(* CODESYS project PiecuchProjekt.export

Project tree, tasks and I/O mapping:
  Device : CODESYS Control Win V3, 3S - Smart Software Solutions GmbH, version 3.5.16.40
    application Application
      libraries: Standard, * (System)
      task MainTask (cyclic, interval t#20ms, priority 1) calls PLC_PRG
      global variables HMI
      global variables OPC
      program PLC_PRG [ST]
      function block TwoAxisLogic [ST]
*)

// Device/Application/HMI
{attribute 'qualified_only'}
VAR_GLOBAL
	GoingQA : BOOL;
	Emitter1Color : INT;
	Emitter2Color : INT;
END_VAR

// Device/Application/OPC
{attribute 'qualified_only'}
VAR_GLOBAL
	// This part includes 2 first machines center and surroundings machines
	iAtAssembledConvEntry : BOOL;
	iAtAssemledPosition : BOOL;
	iMachine1Exit : BOOL;
	iMachine2Exit : BOOL;
	iMachine1Entry : BOOL;
	iMachine2Entry : BOOL;
	iMachiningCenter1Error : BOOL;
	iMachiningCenter2Error : BOOL;
	iMachiningCenter1IsBusy : BOOL;
	iMachiningCenter1Opened : BOOL;
	iMachiningCenter2IsBusy : BOOL;
	iMachiningCenter2Opened : BOOL;
	iMachiningCenter1Progress : INT;
	iMachiningCenter2Progress : INT;
	iRightPositioner2Clamped : BOOL;
	iRightPositioner1Clamped : BOOL;
	iRightPositioner1OnPlace : BOOL;
	iRightPositioner2OnPlace : BOOL;
	iRightPositioner3Clamped : BOOL;
	iRightPositioner3OnPlace : BOOL;
	iTwoAxis1Grabbed : BOOL;
	iTwoAxis1MovingX : BOOL;
	iTwoAxis1MovingZ : BOOL;
	iVisionSenserPart1 : INT;
	iVisionSenserPart2 : INT;
	
	oAssembledMaterialConv : BOOL;
	oBaseMaterialConv1 : BOOL;
	oBaseMaterialConv2 : BOOL;
	oEmitter1Base : INT;
	oEmitter1Emit : BOOL;
	oEmitter1Part : INT;
	oEmitter2Base : INT;
	oEmitter2Emit : BOOL;
	oEmitter2Part : INT;
	oLiquidMaterialConv1 : BOOL;
	oLiquidMaterialConv2 : BOOL;
	oMachiningCenter1Product : BOOL;
	oMachiningCenter2Product : BOOL;
	oRawMaterialSupply1 : BOOL;
	oRawMaterialSupply2 : BOOL;
	oRightPositioner2Clamp : BOOL;
	oRightPositioner1Clamp : BOOL;
	oRightPositioner1Raise : BOOL;
	oRightPositioner2Raise : BOOL;
	oRightPositioner3Clamp : BOOL;
	oRightPositioner3Raise : BOOL;
	oTwoAxis1X : BOOL;
	oTwoAxis1Z : BOOL;
	oTwoAxis1Grab : BOOL;
	
	//This part include second and third twoAxis pick and place, QA and surroundings conveyors, and first warehouse conveyros
	iAtAssemblyLoadEntry : BOOL;
	iAtCrane1Entry : BOOL;
	iAtCurveConv1Exit : BOOL;
	iAtCurveConv1Entry : BOOL;
	iAtFirstwarehouseCurveConv2Exit : BOOL;
	iAtFirstwarehouseCurveConv2Entry : BOOL;
	iAtPusher : BOOL;
	iAtQACurveEntry : BOOL;
	iAtQAEntry : BOOL;
	iAtQAExit : BOOL;
	iAtWeightConvExit : BOOL;
	iAtWeightConvEntry : BOOL;
	iAtTurntable1Entry : BOOL;
	iAtTurntable1ExitQA : BOOL;
	iAtTurntable1ExitNormal : BOOL;
	iPusher1Back : BOOL;
	iPusher2Back : BOOL;
	iPusher3Back : BOOL;
	iPusher1Front : BOOL;
	iPusher2Front : BOOL;
	iPusher3Front : BOOL;
	iTurntable1Back : BOOL;
	iTurntable1Front : BOOL;
	iTurntable1AtZero : BOOL;
	iTurntable1AtNinety : BOOL;
	iTwoAxis2Grabbed : BOOL;
	iTwoAxis2MovingX : BOOL;
	iTwoAxis3Grabbed : BOOL;
	iTwoAxis3MovingX : BOOL;
	iTwoAxis3MovingZ : BOOL;
	iTwoAxis2MovingZ : BOOL;
	iVisionSensor1 : BOOL;
	iVisionSensor2 : BOOL;
	iWeightConv : REAL;
	iAtQALightConvExit : BOOL;
	
	oFirstWarehouseConv1 : BOOL;
	oFirstWarehouseConv3 : BOOL;
	oFirstWarehouseConvLoad : BOOL;
	oFirstWarehouseCurveConv2 : BOOL;
	oPalletAndBoxConv1 : BOOL;
	oPalletAndBoxConv3 : BOOL;
	oPalletAndBoxCurveConv2 : BOOL;
	oPusher1 : BOOL;
	oPusher2 : BOOL;
	oPusher3 : BOOL;
	oQAConv : BOOL;
	oQACurveConv : BOOL;
	oQALightConv1 : BOOL;
	oQALightConv2 : BOOL;
	oQALightConv3 : BOOL;
	oQALightConv4 : BOOL;
	oTurntable1Turn : BOOL;
	oTurntable1Forward : BOOL;
	oTurntable1Backward : BOOL;
	oTwoAxis2X : BOOL;
	oTwoAxis2Z : BOOL;
	oTwoAxis3X : BOOL;
	oTwoAxis3Z : BOOL;
	oTwoAxis2Grab : BOOL;
	oTwoAxis3Grab : BOOL;
	oWeightConvBackward : BOOL;
	oWeightConvToward : BOOL;
	
	//This part includes two cranes and conveyor betweeen them
	iAtCrane1Exit : BOOL;
	iAtCrane2Exit : BOOL;
	iAtExitWarehouseExit : BOOL;
	iAtTurntable2Exit : BOOL;
	iAtTurntable2Entry : BOOL;
	iAtTurntable2ExitWarehouse1 : BOOL;
	iAtTurntable2ExitWarehouse2 : BOOL;
	iCrane1MovingX : BOOL;
	iCrane1MovingZ : BOOL;
	iCrane2MovingX : BOOL;
	iCrane2MovingZ : BOOL;
	iCrane1MidLimit : BOOL;
	iCrane2MidLimit : BOOL;
	iCrane1LeftLimit : BOOL;
	iCrane2LeftLimit : BOOL;
	iCrane1RightLimit : BOOL;
	iCrane2RightLimit : BOOL;
	iTurntable2Back : BOOL;
	iTurntable2Front : BOOL;
	iTurntable2Atzero : BOOL;
	iTurntable2AtNinety : BOOL;
	
	oCrane1Left : BOOL;
	oCrane1Lift : BOOL;
	oCrane2Left : BOOL;
	oCrane2Lift : BOOL;
	oCrane1Right : BOOL;
	oCrane2Right : BOOL;
	oCrane1TargetPosition : INT;
	oCrane2TargetPosition : INT;
	oExitWarehouseConv1 : BOOL;
	oExitWarehouseConv2 : BOOL;
	oFirstWarehouseConvLoadOpposite : BOOL;
	oSecondWarehouseLoadConvOpposite : BOOL;
	oTowardFirstWarehouse : BOOL;
	oTowardSecondWarehouse : BOOL;
	oTurntable2Turn : BOOL;
	oTurntable2Forward : BOOL;
	oTurntable2Backward : BOOL;

	//this part include Box Pick and Place, and conveyors till elevator
	iAtBoxSupplyCurveConv2Exit : BOOL;
	iAtBoxSupplyCurveConv2Entry : BOOL;
	iAtBoxSupplyEnter : BOOL;
	iAtElevatorEntry : BOOL;
	iAtLoadEmptyBoxEntry : BOOL;
	iAtLoadEmptyBoxExit : BOOL;
	iAtPalletDestinationEntry : BOOL;
	iAtPalletDestinationExit : BOOL;
	iAtSecondWarehouseCurveConv3Exit : BOOL;
	iAtSecondWarehouseCurveConv3Entry : BOOL;
	iBigBox : BOOL;
	iMidBox : BOOL;
	iPickPlace1Rotated : BOOL;
	iPickPlace1CurrentX : REAL;
	iPickPlace1CurrentY : REAL;
	iPickPlace1CurrentZ : REAL;
	iPickPlace1BoxDetected : BOOL;
	iSmallBox : BOOL;
	
	oBoxSupplyConv1 : BOOL;
	oBoxSupplyConv3 : BOOL;
	oBoxSupplyCurveConv2 : BOOL;
	oEmptyBoxConvSupply : BOOL;
	oPickPlace1X : REAL;
	oPickPlace1Y : REAL;
	oPickPlace1Z : REAL;
	oPickPlace1Grab : BOOL;
	oPickPlace1Rotate : BOOL;
	oSecondWarehouseConv1 : BOOL;
	oSecondWarehouseConv2 : BOOL;
	oSecondWarehouseConv4 : BOOL;
	oSecondWarehouseConv5 : BOOL;
	oSecondWarehouseCurveConv3 : BOOL;
	
	//Palletizer
	iAtElevatorUpEntry : BOOL;
	iAtPalletizerChainEntry : BOOL;
	iAtPalletizerConvEntry : BOOL;
	iAtPalletizerEntry : BOOL;
	iPalletizer1Clamped : BOOL;
	iPalletizer1Opening : BOOL;
	iPalletizer1Pushing : BOOL;
	iPalletizer1ElevatorBack : BOOL;
	iPalletizer1ElevatorFront : BOOL;
	iPalletizer1ElevatorMoving : BOOL;
	
	oPalletizer1Open : BOOL;
	oPalletizer1Push : BOOL;
	oPalletizer1Turn : BOOL;
	oPalletizer1Clamp : BOOL;
	oPalletizer1Forward : BOOL;
	oPalletizer1Backward : BOOL;
	oPalletizer1ElevatorUp : BOOL;
	oPalletizer1ChainForward : BOOL;
	oPalletizer1ElevatorDown : BOOL;
	oPalletizer1ChainBackward : BOOL;
	oPalletizer1ElevatorMoveToMax : BOOL;
	oPalletizerConv : BOOL;
	oPalletizerSupplyConv : BOOL;
	oPalletizerSupplyLightConv : BOOL;
	oPalletsTowardElevator : BOOL;
	
	//Elevator
	iAtCrane2Entry : BOOL;
	iAtElevatorExit : BOOL;
	iElevator1LeftLimit : BOOL;
	iElevator1RightLimit : BOOL;
	iElevator1CurrentPoint : REAL;
	oElevator1Forward : BOOL;
	oElevator1Backward : BOOL;
	oElevator1SetPoint : REAL;
	oSecondWarehouseConv6 : BOOL;
	oSecondWarehouseLoadConv : BOOL;
	
	// Control panel Box Supply
	iBoxSupplyAutomatic : BOOL;
	iBoxSupplyEmergency : BOOL;
	iBoxSupplyManual : BOOL;
	iBoxSupplyReset : BOOL;
	iBoxSupplyStart : BOOL;
	iBoxSupplyStop : BOOL;
	iSafetyDoorBoxSupply : BOOL;
	oBoxSupplyDisplay : REAL;
	oBoxSupplyReset : BOOL;
	oBoxSupplyStart : BOOL;
	oBoxSupplyStop : BOOL;
	
	// Control panel palletizer
	iPalletizerAutomatic : BOOL;
	iPalletizerEmergency : BOOL;
	iPalletizerManual : BOOL;
	iPalletizerReset : BOOL;
	iPalletizerStart : BOOL;
	iPalletizerStop : BOOL;
	oPalletizerDisplay : REAL;
	oPalletizerReset : BOOL;
	oPalletizerStart : BOOL;
	oPalletizerStop : BOOL;
	
	// Machine center 1 & 2
	oMachiningCenter1Stop : BOOL;
	oMachiningCenter2Stop : BOOL;
	oMachiningCenter1Reset : BOOL;
	oMachiningCenter1Start : BOOL;
	oMachiningCenter2Reset : BOOL;
	oMachiningCenter2Start : BOOL;
	
	// Control panel Assembly
	iAssemblyAutomatic : BOOL;
	iAssemblyEmergency : BOOL;
	iAssemblyManual : BOOL;
	iAssemblyReset : BOOL;
	iAssemblyStart : BOOL;
	iAssemblyStop : BOOL;
	oAssemblyDisplay : REAL;
	oAssemblyReset : BOOL;
	oAssemblyStart : BOOL;
	oAssemblyStop : BOOL;
	
END_VAR

// Device/Application/PLC_PRG
PROGRAM PLC_PRG
VAR
	TwoAxis13Array : ARRAY[0..8] OF INT := [1,3,2,1,3,4,0,0];
	TwoAxis2Array  : ARRAY[0..8] OF INT := [2,1,3,4,1,3,0,1];
	QAArray : ARRAY[0..100, 0..2] OF INT;
	MaterialnBox : CTU;
	Timer1Logic : BOOL;
	Timer1 : TON;
	MaterialsPicked : CTU;
	RaisePositioner1 : BOOL;
	QALightConv1 : BOOL;
	QALightConv234 : BOOL;
	Counter1 : CTUD;
	Counter2 : CTUD;
	F_WeightConvEntry : F_TRIG;
	F_WeightConvExit : F_TRIG;
	CurveArray1 : CTUD;
	NotCurveExit : BOOL;
	TwoAxis1 : TwoAxisLogic;
	TwoAxis2 : TwoAxisLogic;
	TwoAxis3 : TwoAxisLogic;
	LiquidMaterialConv1: BOOL;
	BaseMaterialConv1 : BOOL;
	R_MachineCenter1Working : R_TRIG;
	F_PalletEntryTwoAxis2   : F_TRIG;
	R_QAConv   : R_TRIG;
	F_QAEntry : F_TRIG;
	QAConvWorking : BOOL;
	VisionSensor1        : BOOL;
	VisionSensor2        : BOOL;
	AssemblyMaterialMove : BOOL;
	F_VisionSensor1 	 : F_TRIG;
	F_VisionSensor2 	 : F_TRIG;
	F_AssemblyExit 	 	 : F_TRIG;
	F_Turntable1ExitQA 	 : F_TRIG;
	F_Turntable1ExitNormal : F_TRIG;
	R_Turntable1Front    : R_TRIG;
	Turn1Logic 			 : BOOL;
	TwoAxis1Working 	 : BOOL;
	TwoAxis2Working		 : BOOL;
	TwoAxis3Working 	 : BOOL;
	TwoAxis2WorkingPosition : BOOL;
	TwoAxis2MaterialReady : BOOL;
	TwoAxis3WorkingPosition : BOOL;
	Part1Ready : BOOL;
	Part2Ready : BOOL;
	Clamping1 : BOOL;
	Clamping2 : BOOL;
	Clamping3 : BOOL;
	TwoAxis1MoveDown : BOOL;
	TwoAxis1MoveUp : BOOL;
	TwoAxis1MoveForward : BOOL;
	TwoAxis1MoveBackward : BOOL;
	TwoAxis1Grabbed : BOOL;
	TwoAxis1Done : BOOL;
	AssemblyConvMove : BOOL;
	F_AssembledPosition : F_TRIG;
	PalletAndBoxConv3 : BOOL;
	Turntable1Forward : BOOL;
	
END_VAR

(* Logic behind Machine Center 1 *)

// Emitter should always be true, changing it's color will be done from HMI
OPC.oEmitter1Emit := TRUE;
OPC.oEmitter1Part := HMI.Emitter1Color;
// Conv supply should send raw material only when machine 1 center not busy and there is no raw material at entry
OPC.oRawMaterialSupply1 := NOT OPC.iMachine1Entry AND NOT OPC.iMachiningCenter1IsBusy;
// Machine Center should start working as soon as there is raw material in
OPC.oMachiningCenter1Start := OPC.iMachine1Entry;

(* Logic behind Machine Center 2 *)

// Emitter should always be true, changing it's color will be done from HMI
OPC.oEmitter2Emit := TRUE;
OPC.oEmitter2Part := HMI.Emitter2Color;
// We want to make second part of material so we must change this variable to true
OPC.oMachiningCenter2Product := TRUE;
// Conv supply should send raw material only when machine 2 center not busy and there is no raw material at entry
OPC.oRawMaterialSupply2 := NOT OPC.iMachine2Entry AND NOT OPC.iMachiningCenter2IsBusy;
// Machine Center should start working as soon as there is raw material in
OPC.oMachiningCenter2Start := OPC.iMachine2Entry;

(* Converoys from Machine center *)

// At first we want to make CTUD counter which will count how many parts are in move
Counter1(CU := OPC.iMachine1Exit, CD:= VisionSensor1);
Counter2(CU := OPC.iMachine2Exit, CD:= VisionSensor2);

// Now when we have our counter, if the CV is bigger than 0, QD whille be false so we have mocing part
LiquidMaterialConv1 := NOT Counter2.QD;

// Same as above, if CV bigger than 0, conv should move if possible
BaseMaterialConv1 := NOT Counter1.QD;

// When should move conveyors from machine center 2
OPC.oLiquidMaterialConv1 := OPC.oLiquidMaterialConv2 AND LiquidMaterialConv1 ;
OPC.oLiquidMaterialConv2 := NOT TwoAxis1Working OR AssemblyMaterialMove;

// When should move conveyors from machine center 1
OPC.oBaseMaterialConv1 := OPC.oBaseMaterialConv2 AND BaseMaterialConv1 ;
OPC.oBaseMaterialConv2 := NOT TwoAxis1Working;

(* Two Axis Pick & Place which assemble two parts, two vision sensors, two right positioners and  light conv behind them *)

// At first we want to make falling trigger using vision senser, those numbers are taken from factory i/o
IF OPC.iVisionSenserPart1 = 572 OR OPC.iVisionSenserPart1 = 580 OR OPC.iVisionSenserPart1 = 588 THEN
	VisionSensor1 := TRUE;
ELSE 
	VisionSensor1 := FALSE;
END_IF;

// Same as previous we want to check when expected material went in
IF OPC.iVisionSenserPart2 = 562 OR OPC.iVisionSenserPart2 = 563 OR OPC.iVisionSenserPart2 = 564 THEN
	VisionSensor2 := TRUE;
ELSE 
	VisionSensor2 := FALSE;
END_IF;

// Making falling trigger 
F_VisionSensor1(CLK := VisionSensor1);
F_VisionSensor2(CLK := VisionSensor2);

// Checking if the parts are on positon, then clamping them
IF F_VisionSensor1.Q THEN 
	Clamping1 := TRUE;
	OPC.oRightPositioner1Clamp := TRUE;
END_IF;

// Checking if clamped
IF Clamping1 AND OPC.iRightPositioner1Clamped THEN
	Part1Ready := TRUE;
	OPC.oRightPositioner1Clamp := FALSE;
END_IF;

// Now the very same thing for second positioner

// Checking if the parts are on positon, then clamping them
IF F_VisionSensor2.Q THEN 
	Clamping2 := TRUE;
	OPC.oRightPositioner2Clamp := TRUE;
END_IF;

// Checking if clamped
IF Clamping2 AND OPC.iRightPositioner2Clamped THEN
	Part2Ready := TRUE;
	OPC.oRightPositioner2Clamp := FALSE;
END_IF;

// If both parts are ready, two axis pick and place will assembly them, at first it will move down to take first part
IF Part1Ready AND Part2Ready THEN
	TwoAxis1Working := TRUE;
	Part2Ready := FALSE;
	Part1Ready := FALSE;
END_IF;

// Using FB to pick and plice material
TwoAxis1( Start:= TwoAxis1Working, IncomingArray := TwoAxis13Array, Grabbed := OPC.iTwoAxis1Grabbed, MovingX := OPC.iTwoAxis1MovingX, MovingZ := OPC.iTwoAxis1MovingZ);
OPC.oTwoAxis1X := TwoAxis1.X;
OPC.oTwoAxis1Z := TwoAxis1.Z;
OPC.oTwoAxis1Grab := TwoAxis1.Grab;

// Set working variable to 0 and raise the positioner
IF TwoAxis1.JobDone THEN
	TwoAxis1Working := FALSE;
	RaisePositioner1 := TRUE;
END_IF;

// IF assemby done, then open right positioner 2
OPC.oRightPositioner1Raise := RaisePositioner1;

// When right positioner is up, move material
IF RaisePositioner1 AND  OPC.iRightPositioner1OnPlace THEN
	AssemblyMaterialMove := TRUE;
END_IF;

// Close opened right positioner 2
F_AssemblyExit(CLK := OPC.iAtAssembledConvEntry);
IF F_AssemblyExit.Q THEN
	OPC.oRightPositioner1Raise := FALSE;
	AssemblyMaterialMove := FALSE;
	AssemblyConvMove := TRUE;
	RaisePositioner1 := FALSE;
END_IF;

// Falling trigger at the end of this conv
F_AssembledPosition(CLK := OPC.iAtAssemledPosition);

// When f_trig at the end, stop conveyor
IF F_AssembledPosition.Q THEN
	AssemblyConvMove := FALSE;
	Clamping3 := TRUE;
	OPC.oRightPositioner3Clamp := TRUE;
END_IF;

// Clamp material to desired position
IF Clamping3 AND OPC.iRightPositioner3Clamped THEN
	Clamping3 := FALSE;
	TwoAxis2MaterialReady := TRUE;
	OPC.oRightPositioner3Clamp := FALSE;
END_IF;

// Logic when should this conv move
OPC.oAssembledMaterialConv := AssemblyConvMove ;

(* Logic when should second pick and place take the assembled material *)

//Making rising triggerws which will inform us weather there is pallet in determined place
F_PalletEntryTwoAxis2(CLK := OPC.iAtAssemblyLoadEntry);
// When pallet is on place we set two axis pick place in working stance, now we wait for materials
IF F_PalletEntryTwoAxis2.Q THEN
	TwoAxis2WorkingPosition := TRUE;
END_IF;
// At first we have to move coveroy which send the pallet wuth the box, we usually want it to run when there is no pallet on determined place
OPC.oPalletAndBoxConv1 := NOT TwoAxis2WorkingPosition;

// When should two axis 2 work 
IF TwoAxis2WorkingPosition AND TwoAxis2MaterialReady THEN
	TwoAxis2Working := TRUE;
	TwoAxis2MaterialReady := FALSE;
END_IF;

// Calling FB which will take the element and place it in the box
TwoAxis2( Start:= TwoAxis2Working, IncomingArray := TwoAxis2Array, Grabbed := OPC.iTwoAxis2Grabbed, MovingX := OPC.iTwoAxis2MovingX, MovingZ := OPC.iTwoAxis2MovingZ);
OPC.oTwoAxis2X := TwoAxis2.X;
OPC.oTwoAxis2Z := TwoAxis2.Z;
OPC.oTwoAxis2Grab := TwoAxis2.Grab;


// When job is done we set variable back to 0
IF TwoAxis2.JobDone THEN
	TwoAxis2Working := FALSE;
END_IF;

// Now we would like to count how many things we have in box
MaterialnBox(CU := TwoAxis2.JobDone, PV := 3);

// If we've got 3 materials in box we set the box out
IF MaterialnBox.Q THEN
	MaterialnBox.RESET := MaterialnBox.Q;
	TwoAxis2WorkingPosition := FALSE;
END_IF;

(* This part is about sending box either to QA or Magazine *)

// We would like to use counter in order to power conveyor, but cu and cd require raising trigger so we need to invert one variable
NotCurveExit := NOT OPC.iAtCurveConv1Exit;

// Counter
CurveArray1(CU := OPC.iAtCurveConv1Entry, CD:= NotCurveExit);

// If there is more than one pallet, simply power the curve conveyor
OPC.oPalletAndBoxCurveConv2 := NOT CurveArray1.QD;


// Long conv before first turntable
IF OPC.iAtCurveConv1Exit THEN
	PalletAndBoxConv3 := TRUE;
END_IF

// When should move conveoyr before turn table 1
OPC.oPalletAndBoxConv3 := PalletAndBoxConv3 AND(NOT OPC.iAtTurntable1Entry OR OPC.iTurntable1AtZero);

// Move pallet to the middle of turn table
IF OPC.iAtTurntable1Entry THEN
	Turntable1Forward := TRUE;
END_IF;

// If at middle, set to false both conveyros and turn
R_Turntable1Front(CLK := OPC.iTurntable1Front); 

// When package is on the front we want to stop conveyors and rotate it
IF R_Turntable1Front.Q THEN
	Turntable1Forward := FALSE;
	PalletAndBoxConv3 := FALSE;
	Turn1Logic := TRUE;
END_IF

// Tabl;e should turn when rising trigger fornt sensor
OPC.oTurntable1Turn := Turn1Logic;

// Making 2 falling triggers which inform us when pallet lefts table
F_Turntable1ExitQA(CLK := OPC.iAssemblyAutomatic);
F_Turntable1ExitNormal(CLK := OPC.iAtTurntable1ExitNormal);

// IF left turn table, return to normal
IF F_Turntable1ExitQA.Q OR F_Turntable1ExitNormal.Q THEN
	Turn1Logic := FALSE;
END_IF;

// If turned and going to QA, goo left
OPC.oTurntable1Forward := (HMI.GoingQA AND OPC.iTurntable1AtNinety) OR Turntable1Forward;

// If turned and going warehouse, charge right
OPC.oTurntable1Backward := NOT HMI.GoingQA AND OPC.iTurntable1AtNinety;

// Raising trigger to power our conveyor
R_QAConv(CLK := OPC.iAtTurntable1ExitQA);

// IF raising trigger then change variable which move conv
IF R_QAConv.Q THEN
	QAConvWorking := TRUE;
END_IF;

// Conveor moves when QAConvWorking from raising trigger true
OPC.oQAConv := QAConvWorking;

// Falling trigger to stop our conv
F_QAEntry(CLK := OPC.iAtQAEntry);

// When pallet on it;s place, stop it
IF F_QAEntry.Q THEN
	QAConvWorking := FALSE;
	TwoAxis3Working := TRUE;
	TwoAxis3WorkingPosition := TRUE;
END_IF;

// Instance of FB which operate our two axis
TwoAxis3( Start:= TwoAxis3Working, IncomingArray := TwoAxis13Array, Grabbed := OPC.iTwoAxis3Grabbed, MovingX := OPC.iTwoAxis3MovingX, MovingZ := OPC.iTwoAxis3MovingZ);
OPC.oTwoAxis3X := TwoAxis3.X;
OPC.oTwoAxis3Z := TwoAxis3.Z;
OPC.oTwoAxis3Grab := TwoAxis3.Grab;

// Setting counter which will tell us how many material have been picked
MaterialsPicked( CU := TwoAxis3.JobDone, PV := 3);

// If 3 or more materials picked stop working at this moment, pallet will be pushed next with next pallet entry
IF MaterialsPicked.Q THEN
	TwoAxis3WorkingPosition := FALSE;
END_IF;

// When job done set to false, in order to reset pick up cycle
IF TwoAxis3.JobDone THEN
	TwoAxis3Working := FALSE;
	QALightConv1 := TRUE;
END_IF;
 
// when robot should be working and he's not working(which means he finished one run) run it again
IF TwoAxis3WorkingPosition AND NOT TwoAxis3Working THEN
	TwoAxis3Working := TRUE;
END_IF

// Logic when should move first QA conv
OPC.oQALightConv1 := QALightConv1;

// Making falling trigger which tells us when our material enter weight conv
F_WeightConvEntry(CLK := OPC.iAtWeightConvEntry);

// When our material fully enter weight conv we would like to stop it
IF F_WeightConvEntry.Q THEN
	Timer1Logic := TRUE;
	QALightConv1 := FALSE;
END_IF;

// Logic when should weight conv charge forward
OPC.oWeightConvToward := Timer1.Q OR OPC.iAtWeightConvEntry;

// here we would like to save our readings, not sure how right now
IF Timer1.ET > T#1S THEN
	// !!!!!!!!!!!! THIS IS JUST A FILLER, LATER WHEN WE FIGURE OUT HOW TO DO IT WE WILL DO IT
	QAArray[1,1] := 1;
END_IF;

// timer 1, we need to read analog reading when conv doesnt move so we stop conv and after 2s we want to varge forward
Timer1(IN:= Timer1Logic, PT := T#2S);

// falling trigger which tell us when material leaves weight conv
F_WeightConvExit(CLK := OPC.iAtWeightConvExit);

// When material left weight conv simply stop charging forward
IF F_WeightConvExit.Q THEN
	Timer1Logic := FALSE;
	QALightConv234 := TRUE;
END_IF;

OPC.oQALightConv4 := OPC.oQALightConv3 := OPC.oQALightConv2 := QALightConv234;

END_PROGRAM

// Device/Application/TwoAxisLogic
FUNCTION_BLOCK TwoAxisLogic
VAR_INPUT
	Start   : BOOL;
	Grabbed : BOOL;
	MovingX : BOOL;
	MovingZ : BOOL;
	IncomingArray : ARRAY[0..8] OF INT;
END_VAR
VAR_OUTPUT
	X : BOOL;
	Z : BOOL;
	Grab : BOOL;
	JobDone : BOOL;
END_VAR
VAR
	Variable1 : BOOL := FALSE;
	Variable2 : BOOL := FALSE;
	Variable3 : BOOL := FALSE;
	Variable4 : BOOL := FALSE;
	MyIncrement : INT := 0;
END_VAR

IF START THEN
CASE IncomingArray[Myincrement] OF
	0:
		JobDone := TRUE;
	1:
		Z := TRUE;
		IF Movingz THEN
			Variable1 := TRUE;
		END_IF;
		IF Z AND NOT MovingZ AND( MyIncrement = 0 OR MyIncrement = 1 )AND Variable1 THEN
			Grab := TRUE;
		ELSIF Z AND NOT MovingZ AND( MyIncrement = 3 OR MyIncrement = 4 ) AND Variable1 THEN
			Grab := FALSE;
		END_IF;
		IF Grabbed AND (MyIncrement = 0 OR MyIncrement = 1) THEN;
			MyIncrement := MyIncrement + 1;
			Variable1 := FALSE;
		ELSIF NOT Grabbed AND (MyIncrement = 3 OR MyIncrement = 4) THEN
			MyIncrement := MyIncrement + 1;
			Variable1 := FALSE;
		END_IF;
	2:
		X := TRUE;
		IF MovingX THEN
			Variable2 := TRUE;
		END_IF;
		IF X AND NOT MovingX AND Variable2 THEN
			MyIncrement := MyIncrement + 1;
			Variable2 := FALSE;
		END_IF;
	3:
		Z := FALSE;
		IF Movingz THEN
			Variable3 := TRUE;
		END_IF;
		IF NOT Z AND NOT MovingZ AND Variable3 THEN
			MyIncrement := MyIncrement + 1;
			Variable3 := FALSE;
		END_IF;
	4:
		X := FALSE;
		IF MovingX THEN
			Variable4 := TRUE;
		END_IF;
		IF NOT X AND NOT MovingX AND Variable4 THEN
			MyIncrement := MyIncrement + 1;
			Variable4 := FALSE;
		END_IF;
END_CASE
ELSE
	MyIncrement := 0;
	JobDone := FALSE;
END_IF;

END_FUNCTION_BLOCK
